(*Assign adresses to the pfeiffer controllers connected to this serial terminal*)
stPfeiffer_CTRL_LI3K2_PAX_PTM_01[1].iSerialAddress:= 1;
stPfeiffer_CTRL_LI3K2_PAX_PTM_01[1].xEnableComm:= TRUE;
(*Instanitate the Function block for serial communication with Pfeiffer*)
fbPfeifferCom_LI3K2_PAX_PTM_01(astPfeifferControl:= stPfeiffer_CTRL_LI3K2_PAX_PTM_01,
                              astPfeifferStatus:= stPfeiffer_RBK_LI3K2_PAX_PTM_01,
                              SerialRXBuffer:= SerialRXBuffer_LI3K2_K2B_OUT_PTM_01,
                              SerialTXBuffer:= SerialTXBuffer_LI3K2_K2B_OUT_PTM_01);
(*Copy Status Pv's into the PTM structure*)
fb_LI3K2_K2B_OUT_PTM_01.M_Serial_IO(st_Pfeiffer_RBK:= stPfeiffer_RBK_LI3K2_PAX_PTM_01[1],
                            st_Pfeiffer_CTRL:= stPfeiffer_CTRL_LI3K2_PAX_PTM_01[1]);

(*Assign adresses to the pfeiffer controllers connected to this serial terminal*)
stPfeiffer_CTRL_LI4K2_PAX_PTM_01[1].iSerialAddress:= 1;
stPfeiffer_CTRL_LI4K2_PAX_PTM_01[1].xEnableComm:= TRUE;
(*Instanitate the Function block for serial communication with Pfeiffer*)
fbPfeifferCom_LI4K2_PAX_PTM_01(astPfeifferControl:= stPfeiffer_CTRL_LI4K2_PAX_PTM_01,
                              astPfeifferStatus:= stPfeiffer_RBK_LI4K2_PAX_PTM_01,
                              SerialRXBuffer:= SerialRXBuffer_LI4K2_K2B_OUT_PTM_01,
                              SerialTXBuffer:= SerialTXBuffer_LI4K2_K2B_OUT_PTM_01);
(*Copy Status Pv's into the PTM structure*)
fb_LI4K2_K2B_OUT_PTM_01.M_Serial_IO(st_Pfeiffer_RBK:= stPfeiffer_RBK_LI3K2_PAX_PTM_01[1],
                            st_Pfeiffer_CTRL:= stPfeiffer_CTRL_LI3K2_PAX_PTM_01[1]);

// PIP_Gamma Pumps

fb_PC1K1_ZOS_PIP_1(i_stGauge := fb_PC1K1_ZOS_GPI_1.PG, i_xOverrideMode := xSystemOverrideMode1);
fb_MR1K2_SWITCH_PIP_1(i_stGauge := fb_MR1K2_SWITCH_GPI_1.PG, i_xOverrideMode := xSystemOverrideMode1);
fb_TV1K1_PLEG_PIP_1(i_stGauge := fb_TV1K1_PLEG_GPI_1.PG, i_xOverrideMode := xSystemOverrideMode1);
fb_SL1K2_EXIT_PIP_1(i_stGauge := fb_SL1K2_EXIT_GPI_1.PG, i_xOverrideMode := xSystemOverrideMode1);
fb_ST1K2_PPS_PIP_1(i_stGauge := fb_ST1K2_PPS_GPI_1.PG, i_xOverrideMode := xSystemOverrideMode1);
fb_MR2K2_FLAT_PIP_1(i_stGauge := fb_MR2K2_FLAT_GPI_1.PG, i_xOverrideMode := xSystemOverrideMode2);
fb_MR3K2_KBH_PIP_1(i_stGauge := fb_MR3K2_KBH_GPI_1.PG, i_xOverrideMode := xSystemOverrideMode2);
fb_MR4K2_KBV_PIP_1(i_stGauge := fb_MR4K2_KBV_GPI_1.PG, i_xOverrideMode := xSystemOverrideMode2);
fb_TV4K2_PIP_1(i_stGauge := bm_dummy_gauge, i_xOverrideMode := xSystemOverrideMode2);
fb_IM5K2_PPM_PIP_1(i_stGauge := bm_dummy_gauge, i_xOverrideMode := xSystemOverrideMode2);
fb_PA1K2_PIP_1(i_stGauge := bm_dummy_gauge, i_xOverrideMode := xSystemOverrideMode2);
fb_SP1K2_PAX_PIP_1(i_stGauge := fb_ST1K2_PPS_GPI_1.PG, i_xOverrideMode := xSystemOverrideMode1);  //change interlock to SP1K2 GPI once connected

//SIP Pumps
fb_IM2K2_PPM_PIP_1(i_stGauge := bm_dummy_gauge, i_xOverrideMode := xSystemOverrideMode2);
fb_IM3K2_PPM_PIP_1(i_stGauge := bm_dummy_gauge, i_xOverrideMode := xSystemOverrideMode2);
fb_IM4K2_PPM_PIP_1(i_stGauge := bm_dummy_gauge, i_xOverrideMode := xSystemOverrideMode2);
fb_LI2K2_K2A_PIP_1(i_stGauge := bm_dummy_gauge, i_xOverrideMode := xSystemOverrideMode2);
fb_SP2K2_TXAS_PIP_1(i_stGauge := bm_dummy_gauge, i_xOverrideMode := xSystemOverrideMode2);

//Fast shutter Valve Interface
vfs_dummy_gauge.xPRESS_OK := TRUE;
vfs_dummy_gauge.rPRESS := 0.0000001;
fb_TV1K2_VFS_Interface(IG:=fb_TV4K2_GFS_1.IG, iq_stValve=> , Veto_Valve:=fb_MR4K2_KBV_VGC_2.iq_stValve, i_xVAC_FAULT_OK=> );
//TV1K2_VFS_Interface(IG:= fb_TV4K2_GFS_1.IG);


//Interface for KFE VAC SP1K1-ZOS-VGC-2
// Update interlock signals for RIX
fb_RIX_ILK(
    VG	:=	fb_PC1K1_ZOS_PIP_1.q_IG, //fb_PC1K1_ZOS_GCC_1.IG,
    ILK	:=	st_RIX_ILK
);

END_PROGRAM
